SYSTEM System (* System Configuration *)
  (* Standard: 61499-1 *)
  (* Version 0.0, 1/9/2024, Cheyan, Schneider Electric *)
  {SET_ATTRIBUTE(System.Device.FolderPath, EcoRT_0)}
  APPLICATION APP1
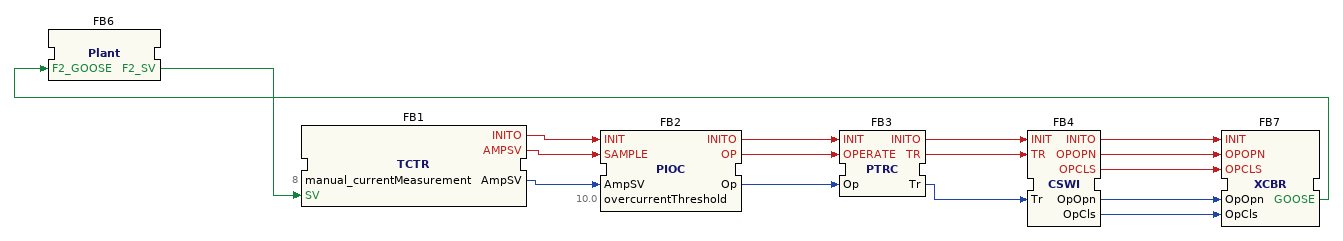
    (* Plant (Power System) *)
    (* Control (IEC 61499) *)
    (* Feeder 2 *)
    FBS
      FB1 : TCTR(manual_currentMeasurement := 8);
      FB6 : Plant;
      FB2 : PIOC(overcurrentThreshold := 10.0);
      FB3 : PTRC;
      FB4 : CSWI;
      FB7 : XCBR;
    END_FBS
    EVENT_CONNECTIONS
      FB1.INITO TO FB2.INIT;
      FB1.AMPSV TO FB2.SAMPLE;
      FB2.INITO TO FB3.INIT;
      FB2.OP TO FB3.OPERATE;
      FB3.INITO TO FB4.INIT;
      FB3.TR TO FB4.TR;
      FB4.INITO TO FB7.INIT;
      FB4.OPOPN TO FB7.OPOPN;
      FB4.OPCLS TO FB7.OPCLS;
    END_CONNECTIONS
    DATA_CONNECTIONS
      FB1.AmpSV TO FB2.AmpSV;
      FB2.Op TO FB3.Op;
      FB3.Tr TO FB4.Tr;
      FB4.OpOpn TO FB7.OpOpn;
      FB4.OpCls TO FB7.OpCls;
    END_CONNECTIONS
    ADAPTER_CONNECTIONS
      FB6.F2_SV TO FB1.SV;
      FB7.GOOSE TO FB6.F2_GOOSE;
    END_CONNECTIONS
  END_APPLICATION
  DEVICE EcoRT_0 : Soft_dPAC
    RESOURCE RES0 : EMB_RES_ECO
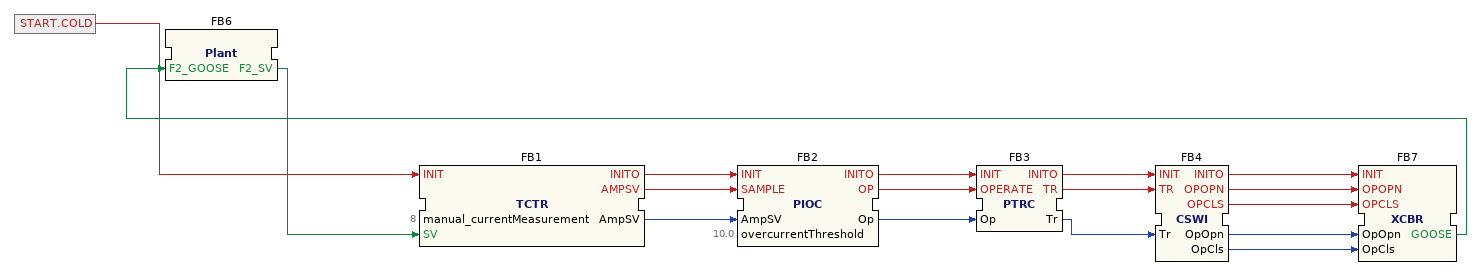
      FBS
        FB6 : Plant;
        FB1 : TCTR(manual_currentMeasurement := 8);
        FB2 : PIOC(overcurrentThreshold := 10.0);
        FB3 : PTRC;
        FB4 : CSWI;
        FB7 : XCBR;
      END_FBS
      EVENT_CONNECTIONS
        FB1.INITO TO FB2.INIT;
        FB1.AMPSV TO FB2.SAMPLE;
        FB2.INITO TO FB3.INIT;
        FB2.OP TO FB3.OPERATE;
        FB3.INITO TO FB4.INIT;
        FB3.TR TO FB4.TR;
        FB4.INITO TO FB7.INIT;
        FB4.OPOPN TO FB7.OPOPN;
        FB4.OPCLS TO FB7.OPCLS;
        START.COLD TO FB1.INIT;
      END_CONNECTIONS
      DATA_CONNECTIONS
        FB1.AmpSV TO FB2.AmpSV;
        FB2.Op TO FB3.Op;
        FB3.Tr TO FB4.Tr;
        FB4.OpOpn TO FB7.OpOpn;
        FB4.OpCls TO FB7.OpCls;
      END_CONNECTIONS
      ADAPTER_CONNECTIONS
        FB6.F2_SV TO FB1.SV;
        FB7.GOOSE TO FB6.F2_GOOSE;
      END_CONNECTIONS
    END_RESOURCE
  END_DEVICE
  MAPPINGS
    APP1.FB6 ON EcoRT_0.RES0;
    APP1.FB1 ON EcoRT_0.RES0;
    APP1.FB2 ON EcoRT_0.RES0;
    APP1.FB3 ON EcoRT_0.RES0;
    APP1.FB4 ON EcoRT_0.RES0;
    APP1.FB7 ON EcoRT_0.RES0;
  END_MAPPINGS
END_SYSTEM
